// TIA Portal V17 export
// export: Created 2023-04-04T13:27:23.8467308Z, ExportSetting WithDefaults, DisplayName Totally Integrated Automation Portal, DisplayVersion V17, DisplayName TIA Portal Openness, DisplayVersion V17, DisplayName TIA Portal Version Control Interface, DisplayVersion V17, DisplayName STEP 7 Professional, DisplayVersion V17, DisplayName STEP 7 Safety, DisplayVersion V17, DisplayName WinCC Advanced, DisplayVersion V17
DATA_BLOCK "gtyp_Interface_Dashboard"   // DB1
TITLE = Global Interface Dashboard Cloud
{ S7_Optimized_Access := 'TRUE' }
AUTHOR : A.Schaefer
VERSION : 0.0
// stored: AutoNumber false, DBAccessibleFromOPCUA true, DBAccessibleFromWebserver true, InstanceOfName typ_MQTT_Interface_Dashboard, InstanceOfType UDT, IsOnlyStoredInLoadMemory false, IsWriteProtectedInAS false
"typ_MQTT_Interface_Dashboard"
   // VAR
   //    Subscribe : "typ_MQTT_Interface_Dashboard_Subscribe";
   //    Publish { S7_SetPoint := 'True'} : "typ_MQTT_ Interface_Dashboard_Publish";
   // END_VAR
BEGIN
END_DATA_BLOCK
